// TIA Portal V19 export
TYPE "MotorAlr"
// stored: Access Published
   STRUCT
      ThermalProtection : Bool;
      Feedback : Bool;
   END_STRUCT;
END_TYPE
